{attribute 'qualified_only'}
{attribute 'strict'}
TYPE Step :
(
	IDLE,
	STARTING,
	HOMING,
	EXECUTE_ZEROING,
	EXECUTE_PICK,
	EXECUTE_PLACE,
	SUSPENDED,
	UNSUSPENDING,
	STOPPED,
	RESETTING

	
);
END_TYPE

(* stored: Version 1.1.0.1, ProductVersion 3.1.4024.12
   DUT Step: Id {58ed28c3-fe9b-46dc-acb8-66d58987fb52} *)
